{attribute 'linkalways'} 
{attribute 'no_explicit_call' := 'This FB is a CLASS and must be accessed using methods or properties'}
{attribute 'enable_dynamic_creation'}
FUNCTION_BLOCK FINAL LT_LINT EXTENDS Node
VAR
	in1 : _LINT(0);
	in2 : _LINT(0);
	out : _BOOL(FALSE);
END_VAR

METHOD PUBLIC Clone : I_Node
VAR
	pNode : POINTER TO LT_LINT;
END_VAR
pNode := __NEW(LT_LINT);
Clone := pNode^;
END_METHOD

METHOD FB_init : BOOL
VAR_INPUT
	bInitRetains : BOOL; // if TRUE, the retain variables are initialized (warm start / cold start)
	bInCopyCode : BOOL;  // if TRUE, the instance afterwards gets moved into the copy code (online change)
END_VAR
AddInput('in1',THIS^.in1);
AddInput('in2',THIS^.in2);
AddOutput('out', THIS^.out);
END_METHOD

METHOD PROTECTED OnExecute
VAR
END_VAR
out.Value := in1.Value < in2.Value;
END_METHOD

END_FUNCTION_BLOCK

(* stored: Version 1.1.0.1, ProductVersion 3.1.4024.15
   POU LT_LINT: Id {71c12f36-aee4-4fc3-9d1a-bc54847da266}, SpecialFunc None
   Folder Constructor: Id {a762d0d4-7e47-44c1-bb5f-d244a054b084}
   Method Clone: Id {b92f3d8c-fa98-429a-bf16-edc87e85db18}
   Method FB_init: Id {3dd975e4-c049-4091-b346-36368619f471}
   Method OnExecute: Id {5695ecf6-2c76-4f80-b461-0ea87aaa843d} *)
